(*
SPDX-FileCopyrightText: Â© 2026 Oleksandr Tiutyk <trofimich@gmail.com>
SPDX-License-Identifier: MIT
License: https://opensource.org/license/mit
*)

(*!
<summary>4-byte union representing raw analog process data.</summary>
<description>
Allows interpreting a 4-byte raw analog signal as signed 16-bit integer, signed 32-bit integer,
or single-precision 32-bit floating point.
</description>
*)

TYPE RAW_ANALOG_VALUE :
UNION
	Int16 : INT;
	Int32 : DINT;
	Real32 : REAL; 
END_UNION
END_TYPE

(* stored: Version 1.1.0.1
   DUT RAW_ANALOG_VALUE: Id {67ca2aae-d8ef-42ae-a8a7-c273fdb3c445} *)
